FUNCTION_BLOCK AIO_OUT (* Service Interface Function Block Type *)
  (* Standard: 61499-2 *)
  (* Version 0.0, 19/05/2021, josef, nxtControl GmBH, template *)
  PACKAGE Flexbridge.Iceblock;
  (* Compiler Cpp nxtControl builtin 1.0 *)
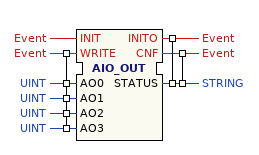
  EVENT_INPUT
    INIT;
    WRITE WITH AO0, AO1, AO2, AO3;
  END_EVENT
  EVENT_OUTPUT
    INITO WITH STATUS;
    CNF WITH STATUS;
  END_EVENT
  VAR_INPUT
    AO0 : UINT;
    AO1 : UINT;
    AO2 : UINT;
    AO3 : UINT;
  END_VAR
  VAR_OUTPUT
    STATUS : STRING; (* Service Status *)
  END_VAR
  SERVICE AIO_OUT/RESOURCE
    SEQUENCE normal_establishment
      AIO_OUT.INIT+(PARAMS) -> RESOURCE.initialize(PARAMS) -> AIO_OUT.INITO+();
    END_SEQUENCE
    SEQUENCE unsuccessful_establishment
      AIO_OUT.INIT+(PARAMS) -> RESOURCE.initialize(PARAMS) -> AIO_OUT.INITO-(STATUS);
    END_SEQUENCE
    SEQUENCE request_confirm
      AIO_OUT.REQ+(SD) -> RESOURCE.request(SD) -> AIO_OUT.CNF+(RD);
    END_SEQUENCE
    SEQUENCE request_inhibited
      AIO_OUT.REQ-(SD) -> AIO_OUT.CNF-(STATUS);
    END_SEQUENCE
    SEQUENCE request_error
      AIO_OUT.REQ+(SD) -> RESOURCE.request(SD) -> AIO_OUT.CNF-(STATUS);
    END_SEQUENCE
    SEQUENCE indication_response
      RESOURCE.indicate(RD) -> AIO_OUT.IND+(RD);
      AIO_OUT.RSP(QI,SD) -> RESOURCE.response(QI,SD);
    END_SEQUENCE
    SEQUENCE indication_inhibited
      RESOURCE.indicate(RD,QI=FALSE) -> RESOURCE.inhibited();
    END_SEQUENCE
    SEQUENCE error_indication
      RESOURCE.error(STATUS) -> AIO_OUT.IND-(STATUS);
    END_SEQUENCE
    SEQUENCE application_initiated_termination
      AIO_OUT.INIT-() -> RESOURCE.terminate() -> AIO_OUT.INITO-(STATUS);
    END_SEQUENCE
    SEQUENCE resource_initiated_termination
      -> AIO_OUT.INITO-(STATUS);
    END_SEQUENCE
  END_SERVICE
END_FUNCTION_BLOCK
